TYPE T_VarInfo : __SYSTEM.VAR_INFO; END_TYPE

(* stored: Version 1.1.0.1, ProductVersion 3.1.4024.14
   DUT T_VarInfo: Id {c31cf113-93e8-018d-198e-e742916a858b} *)
